(* CoDeSys 2.3.9.47 project: Testat2.pro *)
(* Libraries: STANDARD.LIB 5.6.98 11:03:02, C:\Users\Raphael\Documents\HSLU\05_HS_16\ATS\sharedFolder\Projects\Lab_4\lib_lab_4.lib 17.11.16 20:23:40 *)

(* Task configuration *)
TASK Standard (PRIORITY := 0, INTERVAL := T#1ms);
	MAIN
END_TASK

(* POU MAIN, ST *)
PROGRAM MAIN
VAR
(* Variables part A *)
y1 	: REAL := 0;
y2 	: REAL := 0;
y3 	: REAL := 0;
w1	: REAL := 0;
w2	: REAL := 0;
(*Lowpass*)
LP1	:	LowpassFilter;
y4 	:	REAL := 0;



(*Variables part B*)
y5	: REAL := 0;
(*PWM settings*)
duty : REAL := 30; (*DUTY CYCLE*)
peri : REAL := 10; (*SECONDS*)
(*Lowpasses*)
LP2  : LowpassFilter;
LP3  : LowpassFilter;
(**)
y6	 : REAL := 0;

END_VAR
t_cycle := 0.001;
(* Part A *)
(*Sine-Waves*)
w1 := 2*3.1415/5;
w2 := 2*3.1415/0.05;
y1 :=10*SinusFunction(t_global,w1);
y2 :=1*SinusFunction(t_global,w2);
y3 := y1+y2;

(*Lowpassfilter to clear harmonic wave*)
LP1(); LP1.tau := 0.1262; LP1.x_k := y3;

y4 := LP1.y_k;

(* Part B *)
(*PWM*)
y5 := 10*PWMSignal(t_global, duty, peri);


LP2(); LP2.tau := 0.1; LP2.x_k := y5;
LP3(); LP3.tau := 001; LP3.x_k := LP2.y_k;

y6 := LP3.y_k;


(*
(*Integrators*)
INT25(); INT25.e_k := PWMSignal(t_global,25,5);
INT50(); INT50.e_k := PWMSignal(t_global,50,5);
INT75(); INT75.e_k := PWMSignal(t_global,75,5);

LP010(); LP010.tau := 0.1; LP010.x_k := SinusFunction(t_global,10);
LP001(); LP001.tau := 0.1; LP001.x_k := SinusFunction(t_global,1);
LP100(); LP100.tau := 0.1; LP100.x_k := SinusFunction(t_global,100);
(**)

LP010SQ(); LP010SQ.tau := 0.1; LP010SQ.x_k := PWMSignal(t_global,50,(2*3.14)/10);
LP001SQ(); LP001SQ.tau := 0.1; LP001SQ.x_k := PWMSignal(t_global,50,(2*3.14)/1);
LP100SQ(); LP100SQ.tau := 0.1; LP100SQ.x_k := PWMSignal(t_global,50,(2*3.14)/100);

wr := 10*SQRT(1-2*EXPT(0.2,2));
SOL010(); SOL010.w0 := 10; SOL010.d := 0.2;
SOL010.x_k := SinusFunction(t_global,wr/10);

SOL001(); SOL001.w0 := 10; SOL001.d := 0.2;
SOL001.x_k := SinusFunction(t_global,wr/1);


SOL100(); SOL100.w0 := 10; SOL100.d := 0.2;
SOL100.x_k := SinusFunction(t_global,wr*10);
*)

(*Increment Time*)
t_global := t_global + t_cycle;
END_PROGRAM
